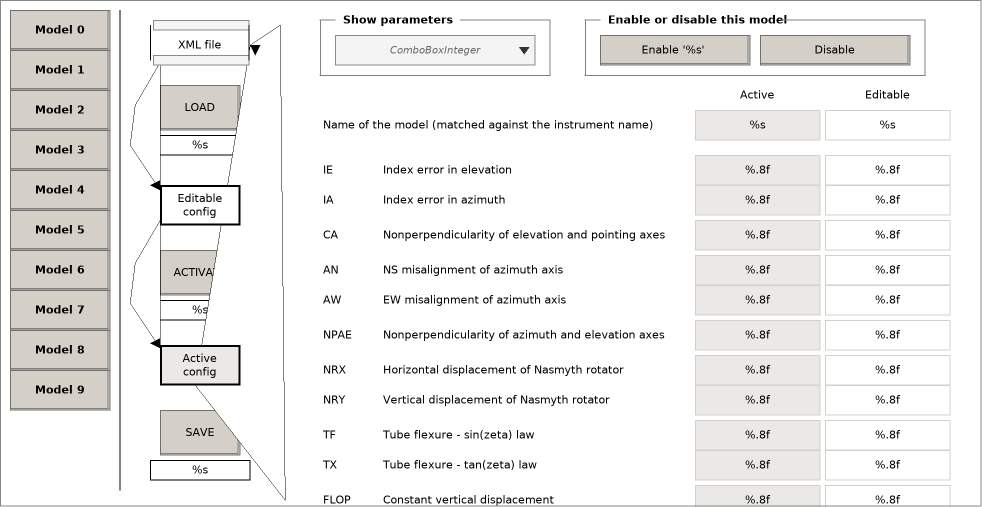
VISUALIZATION VISU_AxesPointingModelsSetup  // 982x507
VAR_IN_OUT
    ref : AxesPointingModelsSetup;
    widget : AxesPointingModelsSetupWidget;
END_VAR
    Button (10,10 100x40), "Model 0", pressed state: widget.activeModel = 0
        OnMouseClick: execute { widget.activeModel := 0; }
    Button (10,50 100x40), "Model 1", pressed state: widget.activeModel = 1
        OnMouseClick: execute { widget.activeModel := 1; }
    Button (10,90 100x40), "Model 2", pressed state: widget.activeModel = 2
        OnMouseClick: execute { widget.activeModel := 2; }
    Button (10,130 100x40), "Model 3", pressed state: widget.activeModel = 3
        OnMouseClick: execute { widget.activeModel := 3; }
    Button (10,170 100x40), "Model 4", pressed state: widget.activeModel = 4
        OnMouseClick: execute { widget.activeModel := 4; }
    Button (10,210 100x40), "Model 5", pressed state: widget.activeModel = 5
        OnMouseClick: execute { widget.activeModel := 5; }
    Button (10,250 100x40), "Model 6", pressed state: widget.activeModel = 6
        OnMouseClick: execute { widget.activeModel := 6; }
    Button (10,290 100x40), "Model 7", pressed state: widget.activeModel = 7
        OnMouseClick: execute { widget.activeModel := 7; }
    Button (10,330 100x40), "Model 8", pressed state: widget.activeModel = 8
        OnMouseClick: execute { widget.activeModel := 8; }
    Button (10,370 100x40), "Model 9", pressed state: widget.activeModel = 9
        OnMouseClick: execute { widget.activeModel := 9; }
    Frame (125,0 855x505), frame switch variable: widget.activeModel
        shows VISU_AxesPointingModelSetup(ref := ref.parts.model0, widget := widget.model0)
        shows VISU_AxesPointingModelSetup(ref := ref.parts.model1, widget := widget.model1)
        shows VISU_AxesPointingModelSetup(ref := ref.parts.model2, widget := widget.model2)
        shows VISU_AxesPointingModelSetup(ref := ref.parts.model3, widget := widget.model3)
        shows VISU_AxesPointingModelSetup(ref := ref.parts.model4, widget := widget.model4)
        shows VISU_AxesPointingModelSetup(ref := ref.parts.model5, widget := widget.model5)
        shows VISU_AxesPointingModelSetup(ref := ref.parts.model6, widget := widget.model6)
        shows VISU_AxesPointingModelSetup(ref := ref.parts.model7, widget := widget.model7)
        shows VISU_AxesPointingModelSetup(ref := ref.parts.model8, widget := widget.model8)
        shows VISU_AxesPointingModelSetup(ref := ref.parts.model9, widget := widget.model9)
    Line (120,490) (120,10)
END_VISUALIZATION

// ---- MTCS/Axes/Visu/VISU_AxesPointDialog.TcVIS
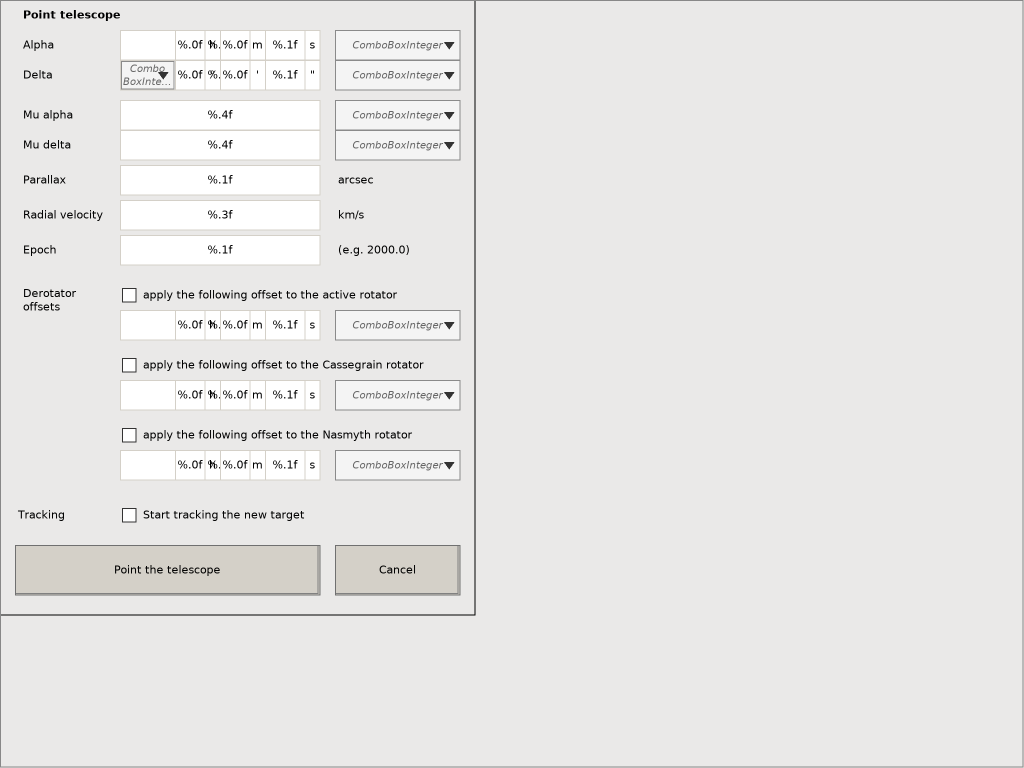
VISUALIZATION VISU_AxesPointDialog  // 1024x768
    Rectangle (0,0 475x615)
    Label (20,5 105x20), "Point telescope"
    Label (20,30 95x30), "Alpha"
    Label (20,60 95x30), "Delta"
    Textfield (120,30 200x30), "%.8f", text variable: GLOBAL.gui.axes.point.field_alpha_decimal, invisible if: GLOBAL.gui.axes.point.units_alpha = AxesDialogAlphaUnits.DIALOG_HMS
        OnMouseClick: write the text variable via VisuDialogs.Numpad
    Textfield (120,60 200x30), "%.8f", text variable: GLOBAL.gui.axes.point.field_delta_decimal, invisible if: GLOBAL.gui.axes.point.units_delta = AxesDialogDeltaUnits.DIALOG_DMS
        OnMouseClick: write the text variable via VisuDialogs.Numpad
    Label (20,100 95x30), "Mu alpha"
    Label (20,130 95x30), "Mu delta"
    Textfield (120,100 200x30), "%.4f", text variable: GLOBAL.gui.axes.point.field_muAlpha
        OnMouseClick: write the text variable via VisuDialogs.Numpad
    Label (20,165 95x30), "Parallax"
    Label (20,200 95x30), "Radial velocity"
    Label (335,200 80x30), "km/s"
    Label (335,165 80x30), "arcsec"
    Textfield (120,130 200x30), "%.4f", text variable: GLOBAL.gui.axes.point.field_muDelta
        OnMouseClick: write the text variable via VisuDialogs.Numpad
    Textfield (120,165 200x30), "%.1f", text variable: GLOBAL.gui.axes.point.field_parallax
        OnMouseClick: write the text variable via VisuDialogs.Numpad
    Textfield (120,200 200x30), "%.3f", text variable: GLOBAL.gui.axes.point.field_radialVelocity
        OnMouseClick: write the text variable via VisuDialogs.Numpad
    Label (20,235 95x30), "Epoch"
    Label (335,235 80x30), "(e.g. 2000.0)"
    Textfield (120,235 200x30), "%.1f", text variable: GLOBAL.gui.axes.point.field_epoch
        OnMouseClick: write the text variable via VisuDialogs.Numpad
    Button (15,545 305x50), "Point the telescope", input disabled if: GLOBAL.mtcs.parts.axes.processes.point.statuses.enabledStatus.disabled
        OnMouseClick: execute { GLOBAL.gui.axes.point.do_request := TRUE; }
        OnMouseClick: CloseDialog Dialog=VISU_AxesPointDialog, Result=OK, NumpadKeypadSet=True
    ComboBoxInteger (335,30 125x30), variable: GLOBAL.gui.axes.point.units_alpha, text list: 'AxesDialogAlphaUnitsTextList'
    ComboBoxInteger (335,60 125x30), variable: GLOBAL.gui.axes.point.units_delta, text list: 'AxesDialogDeltaUnitsTextList'
    ComboBoxInteger (335,100 125x30), variable: GLOBAL.gui.axes.point.units_mu, text list: 'AxesMuUnitsTextList'
    Button (335,545 125x50), "Cancel"
        OnMouseClick: CloseDialog Dialog=VISU_AxesPointDialog, Result=Cancel, NumpadKeypadSet=True
    ComboBoxInteger (335,130 125x30), variable: GLOBAL.gui.axes.point.units_mu, text list: 'AxesMuUnitsTextList'
    Textfield (175,60 30x30), "%.0f", text variable: GLOBAL.gui.axes.point.field_delta_d, invisible if: GLOBAL.gui.axes.point.units_delta <> AxesDialogDeltaUnits.DIALOG_DMS
        OnMouseClick: write the text variable via VisuDialogs.Numpad
    ComboBoxInteger (121,61 53x28), variable: GLOBAL.gui.axes.point.field_delta_sign, invisible if: GLOBAL.gui.axes.point.units_delta <> AxesDialogDeltaUnits.DIALOG_DMS, text list: 'AxesDialogSignTextList'
    Textfield (220,60 30x30), "%.0f", text variable: GLOBAL.gui.axes.point.field_delta_m, invisible if: GLOBAL.gui.axes.point.units_delta <> AxesDialogDeltaUnits.DIALOG_DMS
        OnMouseClick: write the text variable via VisuDialogs.Numpad
    Textfield (265,60 40x30), "%.1f", text variable: GLOBAL.gui.axes.point.field_delta_s, invisible if: GLOBAL.gui.axes.point.units_delta <> AxesDialogDeltaUnits.DIALOG_DMS
        OnMouseClick: write the text variable via VisuDialogs.Numpad
    Label (205,60 15x30), "°", invisible if: GLOBAL.gui.axes.point.units_delta <> AxesDialogDeltaUnits.DIALOG_DMS
    Label (250,60 15x30), "'", invisible if: GLOBAL.gui.axes.point.units_delta <> AxesDialogDeltaUnits.DIALOG_DMS
    Label (305,60 15x30), """, invisible if: GLOBAL.gui.axes.point.units_delta <> AxesDialogDeltaUnits.DIALOG_DMS
    Textfield (175,30 30x30), "%.0f", text variable: GLOBAL.gui.axes.point.field_alpha_h, invisible if: GLOBAL.gui.axes.point.units_alpha <> AxesDialogAlphaUnits.DIALOG_HMS
        OnMouseClick: write the text variable via VisuDialogs.Numpad
    Textfield (220,30 30x30), "%.0f", text variable: GLOBAL.gui.axes.point.field_alpha_m, invisible if: GLOBAL.gui.axes.point.units_alpha <> AxesDialogAlphaUnits.DIALOG_HMS
        OnMouseClick: write the text variable via VisuDialogs.Numpad
    Textfield (265,30 40x30), "%.1f", text variable: GLOBAL.gui.axes.point.field_alpha_s, invisible if: GLOBAL.gui.axes.point.units_alpha <> AxesDialogAlphaUnits.DIALOG_HMS
        OnMouseClick: write the text variable via VisuDialogs.Numpad
    Label (205,30 15x30), "h", invisible if: GLOBAL.gui.axes.point.units_alpha <> AxesDialogAlphaUnits.DIALOG_HMS
    Label (250,30 15x30), "m", invisible if: GLOBAL.gui.axes.point.units_alpha <> AxesDialogAlphaUnits.DIALOG_HMS
    Label (305,30 15x30), "s", invisible if: GLOBAL.gui.axes.point.units_alpha <> AxesDialogAlphaUnits.DIALOG_HMS
    Checkbox (120,500 300x30), "Start tracking the new target", variable: GLOBAL.gui.axes.point.field_tracking
    Label (15,500 95x30), "Tracking"
    Checkbox (120,280 305x30), "apply the following offset to the active rotator", variable: GLOBAL.gui.axes.point.selected_rot, input disabled if: GLOBAL.gui.axes.point.selected_ron OR GLOBAL.gui.axes.point.selected_roc
    Checkbox (120,350 340x30), "apply the following offset to the Cassegrain rotator", variable: GLOBAL.gui.axes.point.selected_roc, input disabled if: GLOBAL.gui.axes.point.selected_rot
    Label (20,280 95x40), "Derotator offsets"
    Textfield (120,310 200x30), "%.8f", text variable: GLOBAL.gui.axes.point.field_rot_decimal, invisible if: GLOBAL.gui.axes.point.units_rot = AxesMoveProcessWidgetUnits.DEGMINSEC, input disabled if: NOT GLOBAL.gui.axes.point.selected_rot
        OnMouseClick: write the text variable via VisuDialogs.Numpad
    ComboBoxInteger (335,310 125x30), variable: GLOBAL.gui.axes.point.units_rot, input disabled if: NOT GLOBAL.gui.axes.point.selected_rot, text list: 'AxesMoveProcessUnitsTextList'
    Textfield (175,310 30x30), "%.0f", text variable: GLOBAL.gui.axes.point.field_rot_d, invisible if: GLOBAL.gui.axes.point.units_rot <> AxesMoveProcessWidgetUnits.DEGMINSEC, input disabled if: NOT GLOBAL.gui.axes.point.selected_rot
        OnMouseClick: write the text variable via VisuDialogs.Numpad
    Textfield (220,310 30x30), "%.0f", text variable: GLOBAL.gui.axes.point.field_rot_m, invisible if: GLOBAL.gui.axes.point.units_rot <> AxesMoveProcessWidgetUnits.DEGMINSEC, input disabled if: NOT GLOBAL.gui.axes.point.selected_rot
        OnMouseClick: write the text variable via VisuDialogs.Numpad
    Textfield (265,310 40x30), "%.1f", text variable: GLOBAL.gui.axes.point.field_rot_s, invisible if: GLOBAL.gui.axes.point.units_rot <> AxesMoveProcessWidgetUnits.DEGMINSEC, input disabled if: NOT GLOBAL.gui.axes.point.selected_rot
        OnMouseClick: write the text variable via VisuDialogs.Numpad
    Label (205,310 15x30), "h", invisible if: GLOBAL.gui.axes.point.units_rot <> AxesMoveProcessWidgetUnits.DEGMINSEC
    Label (250,310 15x30), "m", invisible if: GLOBAL.gui.axes.point.units_rot <> AxesMoveProcessWidgetUnits.DEGMINSEC
    Label (305,310 15x30), "s", invisible if: GLOBAL.gui.axes.point.units_rot <> AxesMoveProcessWidgetUnits.DEGMINSEC
    Checkbox (120,420 335x30), "apply the following offset to the Nasmyth rotator", variable: GLOBAL.gui.axes.point.selected_ron, input disabled if: GLOBAL.gui.axes.point.selected_rot
    Textfield (120,380 200x30), "%.8f", text variable: GLOBAL.gui.axes.point.field_roc_decimal, invisible if: GLOBAL.gui.axes.point.units_rot = AxesMoveProcessWidgetUnits.DEGMINSEC, input disabled if: GLOBAL.gui.axes.point.selected_rot
        OnMouseClick: write the text variable via VisuDialogs.Numpad
    ComboBoxInteger (335,380 125x30), variable: GLOBAL.gui.axes.point.units_rot, input disabled if: GLOBAL.gui.axes.point.selected_rot, text list: 'AxesMoveProcessUnitsTextList'
    Textfield (175,380 30x30), "%.0f", text variable: GLOBAL.gui.axes.point.field_roc_d, invisible if: GLOBAL.gui.axes.point.units_rot <> AxesMoveProcessWidgetUnits.DEGMINSEC, input disabled if: GLOBAL.gui.axes.point.selected_rot
        OnMouseClick: write the text variable via VisuDialogs.Numpad
    Textfield (220,380 30x30), "%.0f", text variable: GLOBAL.gui.axes.point.field_roc_m, invisible if: GLOBAL.gui.axes.point.units_rot <> AxesMoveProcessWidgetUnits.DEGMINSEC, input disabled if: GLOBAL.gui.axes.point.selected_rot
        OnMouseClick: write the text variable via VisuDialogs.Numpad
    Textfield (265,380 40x30), "%.1f", text variable: GLOBAL.gui.axes.point.field_roc_s, invisible if: GLOBAL.gui.axes.point.units_rot <> AxesMoveProcessWidgetUnits.DEGMINSEC, input disabled if: GLOBAL.gui.axes.point.selected_rot
        OnMouseClick: write the text variable via VisuDialogs.Numpad
    Label (205,380 15x30), "h", invisible if: GLOBAL.gui.axes.point.units_rot <> AxesMoveProcessWidgetUnits.DEGMINSEC
    Label (250,380 15x30), "m", invisible if: GLOBAL.gui.axes.point.units_rot <> AxesMoveProcessWidgetUnits.DEGMINSEC
    Label (305,380 15x30), "s", invisible if: GLOBAL.gui.axes.point.units_rot <> AxesMoveProcessWidgetUnits.DEGMINSEC
    Textfield (120,450 200x30), "%.8f", text variable: GLOBAL.gui.axes.point.field_ron_decimal, invisible if: GLOBAL.gui.axes.point.units_rot = AxesMoveProcessWidgetUnits.DEGMINSEC, input disabled if: GLOBAL.gui.axes.point.selected_rot
        OnMouseClick: write the text variable via VisuDialogs.Numpad
    ComboBoxInteger (335,450 125x30), variable: GLOBAL.gui.axes.point.units_rot, input disabled if: GLOBAL.gui.axes.point.selected_rot, text list: 'AxesMoveProcessUnitsTextList'
    Textfield (175,450 30x30), "%.0f", text variable: GLOBAL.gui.axes.point.field_ron_d, invisible if: GLOBAL.gui.axes.point.units_rot <> AxesMoveProcessWidgetUnits.DEGMINSEC, input disabled if: GLOBAL.gui.axes.point.selected_rot
        OnMouseClick: write the text variable via VisuDialogs.Numpad
    Textfield (220,450 30x30), "%.0f", text variable: GLOBAL.gui.axes.point.field_ron_m, invisible if: GLOBAL.gui.axes.point.units_rot <> AxesMoveProcessWidgetUnits.DEGMINSEC, input disabled if: GLOBAL.gui.axes.point.selected_rot
        OnMouseClick: write the text variable via VisuDialogs.Numpad
    Textfield (265,450 40x30), "%.1f", text variable: GLOBAL.gui.axes.point.field_ron_s, invisible if: GLOBAL.gui.axes.point.units_rot <> AxesMoveProcessWidgetUnits.DEGMINSEC, input disabled if: GLOBAL.gui.axes.point.selected_rot
        OnMouseClick: write the text variable via VisuDialogs.Numpad
    Label (205,450 15x30), "h", invisible if: GLOBAL.gui.axes.point.units_rot <> AxesMoveProcessWidgetUnits.DEGMINSEC
    Label (250,450 15x30), "m", invisible if: GLOBAL.gui.axes.point.units_rot <> AxesMoveProcessWidgetUnits.DEGMINSEC
    Label (305,450 15x30), "s", invisible if: GLOBAL.gui.axes.point.units_rot <> AxesMoveProcessWidgetUnits.DEGMINSEC
END_VISUALIZATION

// ---- MTCS/Axes/Visu/VISU_AxesTarget.TcVIS
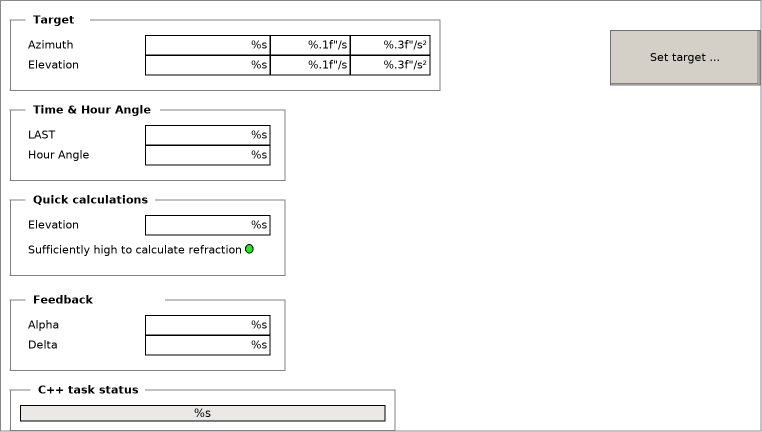
VISUALIZATION VISU_AxesTarget  // 762x432
VAR_IN_OUT
	ref : Axes;
    widget : AxesWidget;
END_VAR
    Polyline (30,390) (10,390) (10,430) (395,430) (395,390) (145,390)
    Rectangle (20,405 365x16), "%s", text variable: widget.cppAxesErrorString
    Label (35,380 115x20), "C++ task status"
    Frame (5,5 390x325)
        shows VISU_AxesFromCpp(ref := ref, widget := widget)
    Button (610,30 150x55), "Set target ..."
        OnMouseClick: OpenDialog Dialog=VISU_AxesSetTargetDialog, OpenModal=True, OpenCentered=True
END_VISUALIZATION

// ---- MTCS/Axes/Visu/VISU_AxesSetTargetDialog.TcVIS
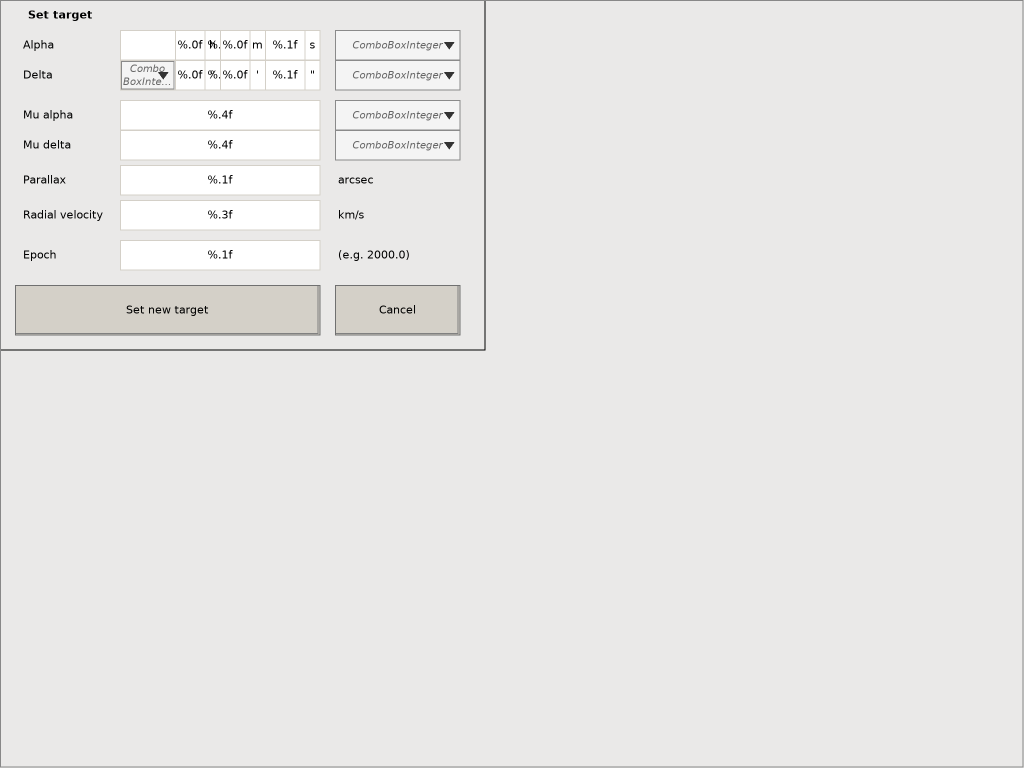
VISUALIZATION VISU_AxesSetTargetDialog  // 1024x768
    Rectangle (0,0 485x350)
    Label (25,5 95x20), "Set target"
    Label (20,30 95x30), "Alpha"
    Label (20,60 95x30), "Delta"
    Textfield (120,30 200x30), "%.8f", text variable: GLOBAL.gui.axes.setTarget.field_alpha_decimal, invisible if: GLOBAL.gui.axes.setTarget.units_alpha = AxesDialogAlphaUnits.DIALOG_HMS
        OnMouseClick: write the text variable via VisuDialogs.Numpad
    Textfield (120,60 200x30), "%.8f", text variable: GLOBAL.gui.axes.setTarget.field_delta_decimal, invisible if: GLOBAL.gui.axes.setTarget.units_delta = AxesDialogDeltaUnits.DIALOG_DMS
        OnMouseClick: write the text variable via VisuDialogs.Numpad
    Label (20,100 95x30), "Mu alpha"
    Label (20,130 95x30), "Mu delta"
    Textfield (120,100 200x30), "%.4f", text variable: GLOBAL.gui.axes.setTarget.field_muAlpha
        OnMouseClick: write the text variable via VisuDialogs.Numpad
    Label (20,165 95x30), "Parallax"
    Label (20,200 95x30), "Radial velocity"
    Label (335,200 80x30), "km/s"
    Label (335,165 80x30), "arcsec"
    Textfield (120,130 200x30), "%.4f", text variable: GLOBAL.gui.axes.setTarget.field_muDelta
        OnMouseClick: write the text variable via VisuDialogs.Numpad
    Textfield (120,165 200x30), "%.1f", text variable: GLOBAL.gui.axes.setTarget.field_parallax
        OnMouseClick: write the text variable via VisuDialogs.Numpad
    Textfield (120,200 200x30), "%.3f", text variable: GLOBAL.gui.axes.setTarget.field_radialVelocity
        OnMouseClick: write the text variable via VisuDialogs.Numpad
    Label (20,240 95x30), "Epoch"
    Label (335,240 80x30), "(e.g. 2000.0)"
    Textfield (120,240 200x30), "%.1f", text variable: GLOBAL.gui.axes.setTarget.field_epoch
        OnMouseClick: write the text variable via VisuDialogs.Numpad
    Button (15,285 305x50), "Set new target", input disabled if: GLOBAL.mtcs.parts.axes.processes.setTarget.statuses.enabledStatus.disabled
        OnMouseClick: execute { GLOBAL.gui.axes.setTarget.do_request := TRUE; }
        OnMouseClick: CloseDialog Dialog=VISU_AxesPointDialog, Result=OK, NumpadKeypadSet=True
    ComboBoxInteger (335,30 125x30), variable: GLOBAL.gui.axes.setTarget.units_alpha, text list: 'AxesDialogAlphaUnitsTextList'
    ComboBoxInteger (335,60 125x30), variable: GLOBAL.gui.axes.setTarget.units_delta, text list: 'AxesDialogDeltaUnitsTextList'
    ComboBoxInteger (335,100 125x30), variable: GLOBAL.gui.axes.setTarget.units_mu, text list: 'AxesMuUnitsTextList'
    Button (335,285 125x50), "Cancel"
        OnMouseClick: CloseDialog Dialog=VISU_AxesSetTargetDialog, Result=Cancel, NumpadKeypadSet=True
    ComboBoxInteger (335,130 125x30), variable: GLOBAL.gui.axes.setTarget.units_mu, text list: 'AxesMuUnitsTextList'
    Textfield (175,60 30x30), "%.0f", text variable: GLOBAL.gui.axes.setTarget.field_delta_d, invisible if: GLOBAL.gui.axes.setTarget.units_delta <> AxesDialogDeltaUnits.DIALOG_DMS
        OnMouseClick: write the text variable via VisuDialogs.Numpad
    ComboBoxInteger (121,61 53x28), variable: GLOBAL.gui.axes.setTarget.field_delta_sign, invisible if: GLOBAL.gui.axes.setTarget.units_delta <> AxesDialogDeltaUnits.DIALOG_DMS, text list: 'AxesDialogSignTextList'
    Textfield (220,60 30x30), "%.0f", text variable: GLOBAL.gui.axes.setTarget.field_delta_m, invisible if: GLOBAL.gui.axes.setTarget.units_delta <> AxesDialogDeltaUnits.DIALOG_DMS
        OnMouseClick: write the text variable via VisuDialogs.Numpad
    Textfield (265,60 40x30), "%.1f", text variable: GLOBAL.gui.axes.setTarget.field_delta_s, invisible if: GLOBAL.gui.axes.setTarget.units_delta <> AxesDialogDeltaUnits.DIALOG_DMS
        OnMouseClick: write the text variable via VisuDialogs.Numpad
    Label (205,60 15x30), "°", invisible if: GLOBAL.gui.axes.setTarget.units_delta <> AxesDialogDeltaUnits.DIALOG_DMS
    Label (250,60 15x30), "'", invisible if: GLOBAL.gui.axes.setTarget.units_delta <> AxesDialogDeltaUnits.DIALOG_DMS
    Label (305,60 15x30), """, invisible if: GLOBAL.gui.axes.setTarget.units_delta <> AxesDialogDeltaUnits.DIALOG_DMS
    Textfield (175,30 30x30), "%.0f", text variable: GLOBAL.gui.axes.setTarget.field_alpha_h, invisible if: GLOBAL.gui.axes.setTarget.units_alpha <> AxesDialogAlphaUnits.DIALOG_HMS
        OnMouseClick: write the text variable via VisuDialogs.Numpad
    Textfield (220,30 30x30), "%.0f", text variable: GLOBAL.gui.axes.setTarget.field_alpha_m, invisible if: GLOBAL.gui.axes.setTarget.units_alpha <> AxesDialogAlphaUnits.DIALOG_HMS
        OnMouseClick: write the text variable via VisuDialogs.Numpad
    Textfield (265,30 40x30), "%.1f", text variable: GLOBAL.gui.axes.setTarget.field_alpha_s, invisible if: GLOBAL.gui.axes.setTarget.units_alpha <> AxesDialogAlphaUnits.DIALOG_HMS
        OnMouseClick: write the text variable via VisuDialogs.Numpad
    Label (205,30 15x30), "h", invisible if: GLOBAL.gui.axes.setTarget.units_alpha <> AxesDialogAlphaUnits.DIALOG_HMS
    Label (250,30 15x30), "m", invisible if: GLOBAL.gui.axes.setTarget.units_alpha <> AxesDialogAlphaUnits.DIALOG_HMS
    Label (305,30 15x30), "s", invisible if: GLOBAL.gui.axes.setTarget.units_alpha <> AxesDialogAlphaUnits.DIALOG_HMS
END_VISUALIZATION

// ---- MTCS/Axes/Visu/VISU_AxesFromCpp.TcVIS
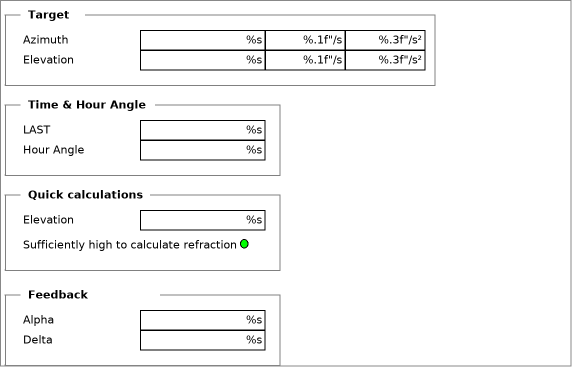
VISUALIZATION VISU_AxesFromCpp  // 572x367
VAR_IN_OUT
	ref : Axes;
    widget : AxesWidget;
END_VAR
    Polyline (20,105) (5,105) (5,175) (280,175) (280,105) (155,105)
    Label (20,120 80x20), "LAST"
    Rectangle (140,120 125x20), "%s", text variable: widget.last.hmsString
    Label (25,95 125x20), "Time & Hour Angle"
    Polyline (20,295) (5,295) (5,365) (280,365) (280,295) (160,295)
    Label (25,285 130x20), "Feedback"
    Label (20,310 105x20), "Alpha"
    Label (20,330 80x20), "Delta"
    Rectangle (140,310 125x20), "%s", text variable: widget.feedback.alpha.hmsString
    Rectangle (140,330 125x20), "%s", text variable: widget.feedback.delta.dmsString
    Label (20,140 80x20), "Hour Angle"
    Rectangle (140,140 125x20), "%s", text variable: widget.ha.hmsString
    Polyline (20,195) (5,195) (5,270) (280,270) (280,195) (150,195)
    Label (25,185 130x20), "Quick calculations"
    Label (20,210 105x20), "Elevation"
    Rectangle (140,210 125x20), "%s", text variable: widget.quickElevation.dmsString
    Frame (0,0 570x85)
        shows VISU_AxesFromCpp_Target(ref := ref, widget := widget)
    Label (20,235 225x20), "Sufficiently high to calculate refraction"
    Frame (240,235 10x15)
        shows VISU_State_green_red(state := ref.target.isTooLow)
END_VISUALIZATION

// ---- MTCS/Axes/Visu/VISU_Axes_Commands_Reset.TcVIS
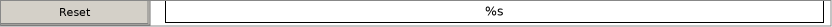
VISUALIZATION VISU_Axes_Commands_Reset  // 832x27
VAR_IN_OUT
    reset : Process;
    resetStatus : StatusWidget;
END_VAR
    Button (0,0 150x25), "Reset", input disabled if: reset.statuses.enabledStatus.disabled
        OnMouseClick: execute { reset.request(); }
    Frame (165,0 665x25)
        shows VISU_StatusWidget(widget := resetStatus)
END_VISUALIZATION

// ---- MTCS/Axes/Visu/VISU_Axes_Commands_Brake.TcVIS
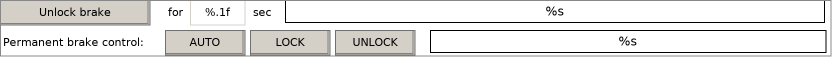
VISUALIZATION VISU_Axes_Commands_Brake  // 832x57
VAR_IN_OUT
    unlockBrake : AxesUnlockBrakeProcess;
    setBrake : SetBrakeProcess;
    unlockBrakeStatus : StatusWidget;
    setBrakeStatus : StatusWidget;
END_VAR
    Button (0,0 150x25), "Unlock brake", input disabled if: unlockBrake.statuses.enabledStatus.disabled
        OnMouseClick: execute { unlockBrake.do_request := TRUE; }
    Frame (285,0 545x25)
        shows VISU_StatusWidget(widget := unlockBrakeStatus)
    Textfield (190,0 55x25), "%.1f", text variable: unlockBrake.set.seconds
        OnMouseClick: write the text variable via VisuDialogs.Numpad
    Label (165,0 30x25), "for"
    Label (245,0 35x25), "sec"
    Button (165,30 80x25), "AUTO", input disabled if: setBrake.statuses.enabledStatus.disabled
        OnMouseClick: execute { setBrake.request(DriveBrakeStates.BRAKE_AUTOMATIC); }
    Button (250,30 80x25), "LOCK", input disabled if: setBrake.statuses.enabledStatus.disabled
        OnMouseClick: execute { setBrake.request(DriveBrakeStates.BRAKE_FORCE_LOCK); }
    Button (335,30 80x25), "UNLOCK", input disabled if: setBrake.statuses.enabledStatus.disabled
        OnMouseClick: execute { setBrake.request(DriveBrakeStates.BRAKE_FORCE_UNLOCK); }
    Frame (430,30 400x25)
        shows VISU_StatusWidget(widget := setBrakeStatus)
    Label (0,30 165x25), "Permanent brake control:"
END_VISUALIZATION

// ---- MTCS/Axes/Visu/VISU_Axes_Commands_Movement.TcVIS
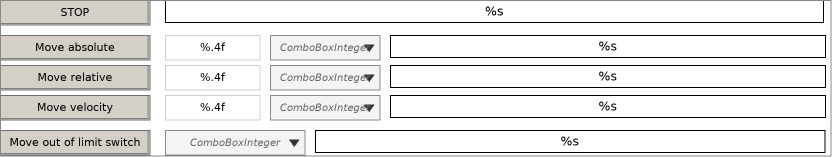
VISUALIZATION VISU_Axes_Commands_Movement  // 832x157
VAR_IN_OUT
    stop : AxesStopProcess;
    moveOutOfLimitSwitch : AxesMoveOutOfLimitSwitchProcess;
    moveAbsolute : AxesMoveAbsoluteProcess;
    moveRelative : AxesMoveRelativeProcess;
    moveVelocity : AxesMoveVelocityProcess;
    
    stopStatus : StatusWidget;
    moveOutOfLimitSwitchStatus : StatusWidget;
    moveAbsoluteStatus : StatusWidget;
    moveRelativeStatus : StatusWidget;
    moveVelocityStatus : StatusWidget;
END_VAR
    Button (0,0 150x25), "STOP", input disabled if: stop.statuses.enabledStatus.disabled
        OnMouseClick: execute { stop.request(); }
    Frame (165,0 665x25)
        shows VISU_StatusWidget(widget := stopStatus)
    Button (0,130 150x25), "Move out of limit switch", input disabled if: moveOutOfLimitSwitch.statuses.enabledStatus.disabled
        OnMouseClick: execute { moveOutOfLimitSwitch.do_request := TRUE; }
    Frame (315,130 515x25)
        shows VISU_StatusWidget(widget := moveOutOfLimitSwitchStatus)
    ComboBoxInteger (165,130 140x25), variable: moveOutOfLimitSwitch.set.switch, text list: 'LimitSwitchesTextList'
    Button (0,35 150x25), "Move absolute", input disabled if: moveAbsolute.statuses.enabledStatus.disabled
        OnMouseClick: execute { moveAbsolute.set.offset := 0.0; moveAbsolute.do_request := TRUE; }
    Textfield (165,35 95x25), "%.4f", text variable: moveAbsolute.set.value
        OnMouseClick: write the text variable via VisuDialogs.Numpad
    ComboBoxInteger (270,35 110x25), variable: moveAbsolute.set.units, text list: 'AxesMoveUnitsTextList'
    Frame (390,35 440x25)
        shows VISU_StatusWidget(widget := moveAbsoluteStatus)
    Button (0,65 150x25), "Move relative", input disabled if: moveRelative.statuses.enabledStatus.disabled
        OnMouseClick: execute { moveRelative.do_request := TRUE; }
    Textfield (165,65 95x25), "%.4f", text variable: moveRelative.set.value
        OnMouseClick: write the text variable via VisuDialogs.Numpad
    ComboBoxInteger (270,65 110x25), variable: moveAbsolute.set.units, text list: 'AxesMoveUnitsTextList'
    Frame (390,65 440x25)
        shows VISU_StatusWidget(widget := moveRelativeStatus)
    Button (0,95 150x25), "Move velocity", input disabled if: moveVelocity.statuses.enabledStatus.disabled
        OnMouseClick: execute { moveVelocity.do_request := TRUE; }
    Textfield (165,95 95x25), "%.4f", text variable: moveVelocity.set.value
        OnMouseClick: write the text variable via VisuDialogs.Numpad
    ComboBoxInteger (270,95 110x25), variable: moveVelocity.set.units, text list: 'AxesMoveVelocityUnitsTextList'
    Frame (390,95 440x25)
        shows VISU_StatusWidget(widget := moveVelocityStatus)
END_VISUALIZATION

// ---- MTCS/Axes/Visu/VISU_Axes_Commands_DoHoming.TcVIS
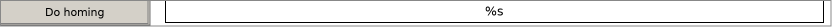
VISUALIZATION VISU_Axes_Commands_DoHoming  // 832x27
VAR_IN_OUT
    doHoming : AxesDoHomingProcess;
    doHomingStatus : StatusWidget;
END_VAR
    Button (0,0 150x25), "Do homing", input disabled if: doHoming.statuses.enabledStatus.disabled
        OnMouseClick: execute { doHoming.request(); }
    Frame (165,0 665x25)
        shows VISU_StatusWidget(widget := doHomingStatus)
END_VISUALIZATION

// ---- MTCS/Axes/Visu/VISU_Axes_stats.TcVIS
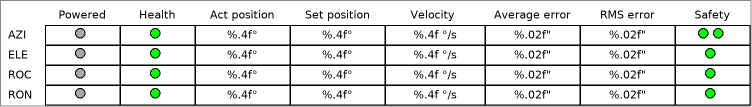
VISUALIZATION VISU_Axes_stats  // 752x107
VAR_IN_OUT
	ref : Axes;
    widget : AxesWidget;
END_VAR
    Rectangle (675,85 75x20)
    Rectangle (675,45 75x20)
    Rectangle (675,65 75x20)
    Rectangle (675,25 75x20)
    Rectangle (45,85 75x20)
    Rectangle (45,45 75x20)
    Rectangle (45,65 75x20)
    Rectangle (45,25 75x20)
    Rectangle (485,25 95x20), "%.02f"", text variable: ref.parts.azi.deviation1SecAverage.arcseconds.value
    Label (485,5 95x20), "Average error"
    Rectangle (580,25 95x20), "%.02f"", text variable: ref.parts.azi.deviation1SecRMS.arcseconds.value
    Rectangle (485,45 95x20), "%.02f"", text variable: ref.parts.ele.deviation1SecAverage.arcseconds.value
    Label (5,25 40x20), "AZI"
    Label (5,45 40x20), "ELE"
    Rectangle (580,45 95x20), "%.02f"", text variable: ref.parts.ele.deviation1SecRMS.arcseconds.value
    Label (580,5 95x20), "RMS error"
    Rectangle (485,65 95x20), "%.02f"", text variable: ref.parts.roc.deviation1SecAverage.arcseconds.value
    Rectangle (580,65 95x20), "%.02f"", text variable: ref.parts.roc.deviation1SecRMS.arcseconds.value
    Rectangle (485,85 95x20), "%.02f"", text variable: ref.parts.ron.deviation1SecAverage.arcseconds.value
    Rectangle (580,85 95x20), "%.02f"", text variable: ref.parts.ron.deviation1SecRMS.arcseconds.value
    Label (5,65 40x20), "ROC"
    Label (5,85 40x20), "RON"
    Label (45,5 75x20), "Powered"
    Frame (75,23 10x15)
        shows VISU_State_gray_green(state := ref.parts.azi.statuses.poweredStatus.enabled)
    Frame (75,43 15x15)
        shows VISU_State_gray_green(state := ref.parts.ele.statuses.poweredStatus.enabled)
    Frame (75,63 10x15)
        shows VISU_State_gray_green(state := ref.parts.roc.statuses.poweredStatus.enabled)
    Frame (75,83 10x15)
        shows VISU_State_gray_green(state := ref.parts.ron.statuses.poweredStatus.enabled)
    Rectangle (195,25 95x20), "%.4f°", text variable: ref.parts.azi.actPos.degrees.value
    Label (195,5 95x20), "Act position"
    Rectangle (195,45 95x20), "%.4f°", text variable: ref.parts.ele.actPos.degrees.value
    Rectangle (195,65 95x20), "%.4f°", text variable: ref.parts.roc.actPos.degrees.value
    Rectangle (195,85 95x20), "%.4f°", text variable: ref.parts.ron.actPos.degrees.value
    Rectangle (385,25 100x20), "%.4f °/s", text variable: ref.parts.azi.actVelo.degreesPerSecond.value
    Label (385,5 95x20), "Velocity"
    Rectangle (385,45 100x20), "%.4f °/s", text variable: ref.parts.ele.actVelo.degreesPerSecond.value
    Rectangle (385,65 100x20), "%.4f °/s", text variable: ref.parts.roc.actVelo.degreesPerSecond.value
    Rectangle (385,85 100x20), "%.4f °/s", text variable: ref.parts.ron.actVelo.degreesPerSecond.value
    Label (675,5 75x20), "Safety"
    Frame (698,23 10x15)
        shows VISU_State_green_red(state := ref.parts.io.parts.aziDrive.parts.channelA.isInSafetate)
    Frame (705,43 15x15)
        shows VISU_State_green_red(state := ref.parts.io.parts.eleDrive.parts.channelA.isInSafetate)
    Frame (705,63 10x15)
        shows VISU_State_green_red(state := ref.parts.io.parts.aziDrive.parts.channelB.isInSafetate)
    Frame (705,83 10x15)
        shows VISU_State_green_red(state := ref.parts.io.parts.ablDrive.parts.channelB.isInSafetate)
    Frame (713,23 10x15)
        shows VISU_State_green_red(state := ref.parts.io.parts.ablDrive.parts.channelA.isInSafetate)
    Rectangle (290,25 95x20), "%.4f°", text variable: ref.parts.azi.setPos.degrees.value
    Label (290,5 95x20), "Set position"
    Rectangle (290,45 95x20), "%.4f°", text variable: ref.parts.ele.setPos.degrees.value
    Rectangle (290,65 95x20), "%.4f°", text variable: ref.parts.roc.setPos.degrees.value
    Rectangle (290,85 95x20), "%.4f°", text variable: ref.parts.ron.setPos.degrees.value
    Rectangle (120,85 75x20)
    Rectangle (120,45 75x20)
    Rectangle (120,65 75x20)
    Rectangle (120,25 75x20)
    Label (120,5 75x20), "Health"
    Frame (150,43 15x15)
        shows VISU_State_green_red(state := ref.parts.ele.statuses.healthStatus.bad)
    Frame (150,63 10x15)
        shows VISU_State_green_red(state := ref.parts.roc.statuses.healthStatus.bad)
    Frame (150,83 10x15)
        shows VISU_State_green_red(state := ref.parts.ron.statuses.healthStatus.bad)
    Frame (150,23 10x15)
        shows VISU_State_green_red(state := ref.parts.azi.statuses.healthStatus.bad)
END_VISUALIZATION

// ---- MTCS/Axes/Widgets/AxesDialogRotUnitsTextList.TcTLO
TEXTLIST AxesDialogRotUnitsTextList
  0 = 'd / m / s'
  1 = 'degrees'
  2 = 'radians'
   = ''
END_TEXTLIST

// ---- MTCS/Axes/Widgets/AxesMoveAlphaDeltaProcessUnitsTextList.TcTLO
TEXTLIST AxesMoveAlphaDeltaProcessUnitsTextList
  0 = 'd/m/s or h/m/s'
  1 = 'degrees'
  2 = 'arcmin'
  3 = 'arcsec'
  4 = 'rad'
   = ''
END_TEXTLIST

// ---- MTCS/Axes/Widgets/AxesDialogAlphaUnitsTextList.TcTLO
TEXTLIST AxesDialogAlphaUnitsTextList
  0 = 'h / m / s'
  1 = 'hours'
  2 = 'radians'
   = ''
END_TEXTLIST

// ---- MTCS/Axes/Widgets/AxesDialogSignTextList.TcTLO
TEXTLIST AxesDialogSignTextList
  0 = '+'
  1 = '-'
   = ''
END_TEXTLIST

// ---- MTCS/Axes/Widgets/AxesMoveUnitsTextList.TcTLO
TEXTLIST AxesMoveUnitsTextList
  0 = 'degrees'
  1 = 'rad'
  2 = 'arcsec'
   = ''
END_TEXTLIST

// ---- MTCS/Axes/Widgets/AxesMoveVelocityUnitsTextList.TcTLO
TEXTLIST AxesMoveVelocityUnitsTextList
  0 = 'degree / s'
  1 = 'arcsec / s'
  2 = 'rad / s'
  3 = 'arcsec / min'
  4 = 'arcsec / hour'
   = ''
END_TEXTLIST

// ---- MTCS/Axes/Widgets/AxesMuUnitsTextList.TcTLO
TEXTLIST AxesMuUnitsTextList
  0 = 'arcsec / year'
  1 = 'mas / year'
  2 = 'deg / year'
  3 = 'rad / year'
   = ''
END_TEXTLIST

// ---- MTCS/Axes/Widgets/AxesDialogDeltaUnitsTextList.TcTLO
TEXTLIST AxesDialogDeltaUnitsTextList
  0 = 'd / m / s'
  1 = 'degrees'
  2 = 'radians'
   = ''
END_TEXTLIST

// ---- MTCS/Axes/Widgets/AxesConfigTextList.TcTLO
TEXTLIST AxesConfigTextList
  0 = 'General'
  1 = 'Known positions'
  2 = 'Location'
  3 = 'Local conditions'
  4 = 'AZI axis (1)'
  5 = 'AZI axis (2)'
  6 = 'AZI axis (3)'
  7 = 'ELE axis (1)'
  8 = 'ELE axis (2)'
  9 = 'ROC axis (1)'
  10 = 'ROC axis (2)'
  11 = 'RON axis (1)'
  12 = 'RON axis (2)'
  13 = 'FW axis'
   = ''
END_TEXTLIST

// ---- MTCS/Axes/Widgets/AxesPointingModelSetupPartsTextList.TcTLO
TEXTLIST AxesPointingModelSetupPartsTextList
  0 = 'Part 1'
  1 = 'Part 2'
   = ''
END_TEXTLIST

// ---- MTCS/Axes/Widgets/AxesMoveProcessUnitsTextList.TcTLO
TEXTLIST AxesMoveProcessUnitsTextList
  0 = 'd / m / s'
  1 = 'degrees'
  2 = 'arcmin'
  3 = 'arcsec'
  4 = 'rad'
   = ''
END_TEXTLIST

// ---- MTCS/Common/Visu/VISU_AX522Drive.TcVIS
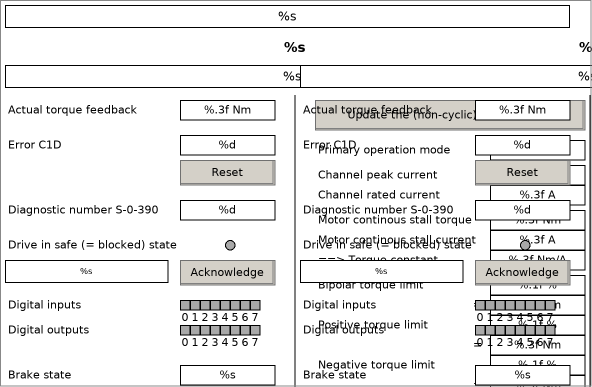
VISUALIZATION VISU_AX522Drive  // 592x387
VAR_IN_OUT
    ref : AX52XXDrive;
    widget : AX52XXDriveWidget;
END_VAR
    Frame (5,5 570x25)
        shows VISU_StatusWidget(widget := widget.actualStatus)
    Frame (0,35 295x350)
        shows VISU_AX522DriveChannel(ref := ref.parts.channelA, widget := widget.channelA)
    Frame (295,35 295x350)
        shows VISU_AX522DriveChannel(ref := ref.parts.channelB, widget := widget.channelB)
END_VISUALIZATION

// ---- MTCS/Common/Visu/VISU_BaseAxis_Gearing.TcVIS
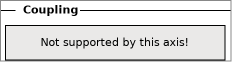
VISUALIZATION VISU_BaseAxis_Gearing  // 232x62
VAR_IN_OUT
	axis : BaseAxis;
    axisWidget : BaseAxisWidget;
END_VAR
    Button (141,25 80x35), "Decouple", input disabled if: axis.processes.gearOut.statuses.enabledStatus.disabled
        OnMouseClick: execute { axis.processes.gearOut.do_request := TRUE; }
    Frame (120,30 20x20)
        shows VISU_State_gray_orange(state := axisWidget.decoupled)
    Button (31,25 80x35), "Couple", input disabled if: axis.processes.gearIn.statuses.enabledStatus.disabled
        OnMouseClick: execute { axis.processes.gearIn.do_request := TRUE; }
    Frame (10,30 25x30)
        shows VISU_State_gray_green(state := axisWidget.coupled)
    Label (20,0 55x20), "Coupling"
    Line (80,10) (230,10)
    Line (0,10) (15,10)
    Rectangle (5,25 220x35), "Not supported by this axis!", invisible if: axis.isGearingSupported
END_VISUALIZATION

// ---- MTCS/Common/Visu/VISU_BaseAxis_MoveVelocity.TcVIS
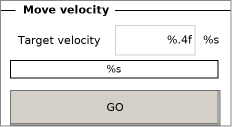
VISUALIZATION VISU_BaseAxis_MoveVelocity  // 232x127
VAR_IN_OUT
	axis : BaseAxis;
    axisWidget : BaseAxisWidget;
    positionSymbol : STRING;
    velocitySymbol : STRING;
END_VAR
    Label (15,26 100x29), "Target velocity"
    Button (10,90 210x35), "GO", input disabled if: axis.processes.moveVelocity.statuses.enabledStatus.disabled
        OnMouseClick: execute { axis.processes.moveVelocity.do_request := TRUE; }
    Line (0,10) (15,10)
    Label (20,0 150x20), "Move velocity"
    Line (115,10) (230,10)
    Textfield (115,25 80x30), "%.4f", text variable: axis.processes.moveVelocity.set.value, input disabled if: axis.processes.moveVelocity.statuses.enabledStatus.disabled
        OnMouseClick: write the text variable via VisuDialogs.Numpad
    Frame (10,60 210x20)
        shows VISU_StatusWidget(widget := axisWidget.moveVelocityProcess.actualStatus)
    Rectangle (200,25 30x30), "%s", text variable: velocitySymbol
END_VISUALIZATION

// ---- MTCS/Common/Visu/VISU_ConfigBOOLEntry_Small.TcVIS
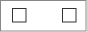
VISUALIZATION VISU_ConfigBOOLEntry_Small  // 87x32
VAR_IN_OUT
    active : BOOL;
    editable : BOOL;
END_VAR
    Checkbox (10,0 45x30), variable: active, input disabled if: TRUE
    Checkbox (60,0 25x30), variable: editable
END_VISUALIZATION

// ---- MTCS/Common/Visu/VISU_ConfigDINTEntry.TcVIS
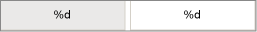
VISUALIZATION VISU_ConfigDINTEntry  // 257x32
VAR_IN_OUT
    active : DINT;
    editable : DINT;
END_VAR
    Textfield (0,0 125x30), "%d", text variable: active, input disabled if: TRUE
    Textfield (130,0 125x30), "%d", text variable: editable, colour toggle: editable <> active
        OnMouseClick: write the text variable via Default
END_VISUALIZATION

// ---- MTCS/Common/Visu/VISU_ConfigREAL4Entry.TcVIS
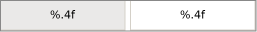
VISUALIZATION VISU_ConfigREAL4Entry  // 257x32
VAR_IN_OUT
    active : REAL;
    editable : REAL;
END_VAR
    Textfield (0,0 125x30), "%.4f", text variable: active, input disabled if: TRUE
    Textfield (130,0 125x30), "%.4f", text variable: editable, colour toggle: editable <> active
        OnMouseClick: write the text variable via Default
END_VISUALIZATION

// ---- MTCS/Common/Visu/VISU_ConfigLREAL8Entry.TcVIS
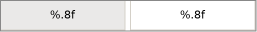
VISUALIZATION VISU_ConfigLREAL8Entry  // 257x32
VAR_IN_OUT
    active : LREAL;
    editable : LREAL;
END_VAR
    Textfield (0,0 125x30), "%.8f", text variable: active, input disabled if: TRUE
    Textfield (130,0 125x30), "%.8f", text variable: editable, colour toggle: editable <> active
        OnMouseClick: write the text variable via Default
END_VISUALIZATION

// ---- MTCS/Common/Visu/VISU_ConfigLREAL1Entry.TcVIS
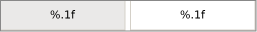
VISUALIZATION VISU_ConfigLREAL1Entry  // 257x32
VAR_IN_OUT
    active : LREAL;
    editable : LREAL;
END_VAR
    Textfield (0,0 125x30), "%.1f", text variable: active, input disabled if: TRUE
    Textfield (130,0 125x30), "%.1f", text variable: editable, colour toggle: editable <> active
        OnMouseClick: write the text variable via Default
END_VISUALIZATION

// ---- MTCS/Common/Visu/VISU_ConfigUINTEntry.TcVIS
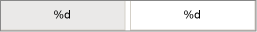
VISUALIZATION VISU_ConfigUINTEntry  // 257x32
VAR_IN_OUT
    active : UINT;
    editable : UINT;
END_VAR
    Textfield (0,0 125x30), "%d", text variable: active, input disabled if: TRUE
    Textfield (130,0 125x30), "%d", text variable: editable, colour toggle: editable <> active
        OnMouseClick: write the text variable via Default
END_VISUALIZATION

// ---- MTCS/Common/Visu/VISU_ConfigBOOLEntry.TcVIS
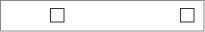
VISUALIZATION VISU_ConfigBOOLEntry  // 205x32
VAR_IN_OUT
    active : BOOL;
    editable : BOOL;
END_VAR
    Checkbox (48,0 45x30), variable: active, input disabled if: TRUE
    Checkbox (178,0 25x30), variable: editable
END_VISUALIZATION

// ---- MTCS/Common/Visu/VISU_ConfigLREAL4Entry.TcVIS
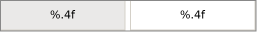
VISUALIZATION VISU_ConfigLREAL4Entry  // 257x32
VAR_IN_OUT
    active : LREAL;
    editable : LREAL;
END_VAR
    Textfield (0,0 125x30), "%.4f", text variable: active, input disabled if: TRUE
    Textfield (130,0 125x30), "%.4f", text variable: editable, colour toggle: editable <> active
        OnMouseClick: write the text variable via Default
END_VISUALIZATION

// ---- MTCS/Common/Visu/VISU_ConfigUDINTEntry.TcVIS
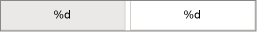
VISUALIZATION VISU_ConfigUDINTEntry  // 257x32
VAR_IN_OUT
    active : UDINT;
    editable : UDINT;
END_VAR
    Textfield (0,0 125x30), "%d", text variable: active, input disabled if: TRUE
    Textfield (130,0 125x30), "%d", text variable: editable, colour toggle: editable <> active
        OnMouseClick: write the text variable via Default
END_VISUALIZATION

// ---- MTCS/Common/Visu/VISU_ConfigINTEntry.TcVIS
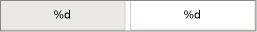
VISUALIZATION VISU_ConfigINTEntry  // 257x32
VAR_IN_OUT
    active : INT;
    editable : INT;
END_VAR
    Textfield (0,0 125x30), "%d", text variable: active, input disabled if: TRUE
    Textfield (130,0 125x30), "%d", text variable: editable, colour toggle: editable <> active
        OnMouseClick: write the text variable via Default
END_VISUALIZATION

// ---- MTCS/Common/Visu/VISU_ConfigUSINTEntry.TcVIS
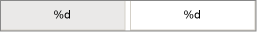
VISUALIZATION VISU_ConfigUSINTEntry  // 257x32
VAR_IN_OUT
    active : USINT;
    editable : USINT;
END_VAR
    Textfield (0,0 125x30), "%d", text variable: active, input disabled if: TRUE
    Textfield (130,0 125x30), "%d", text variable: editable, colour toggle: editable <> active
        OnMouseClick: write the text variable via Default
END_VISUALIZATION

// ---- MTCS/Common/Visu/VISU_CANopenBus.TcVIS
